Omron CX-Programmer project NewProject (CX-Programmer 9.87)

# PLC NewPLC1: CP1L M
; 

## Global symbols (name address type ; comment)
Banco_de_Dados_29 Contador_de_Peças_PH29
Banco_de_Dados_30 Contador_de_Peças_PH30
Banco_de_Dados_31 Contador_de_Peças_PH31
Conta_Peças Contador_de_Peças_PH31
PH11 0.03 BOOL
PH29 0.05 BOOL
PH30 0.04 BOOL
Visual_Formato_Trabalho_29 Formato_de_Trabalho_29
Visual_Formato_Trabalho_30 Formato_de_Trabalho_30
Visual_Formato_Trabalho_31 Formato_de_Trabalho_31
xx Formato_de_Trabalho_29

## Program NuovoProgramma1 (cyclic task 0)
Local symbols
F_31dias_vezes_2_ph30 D546 WORD
F_31dias_vezes_2_ph31 D530 WORD
F_Memoria_contagem_BCD_ph30 D552 WORD
F_Memoria_contagem_BCD_ph31 D536 WORD
F_Memória_de_Armazenagem_ph30 D550 WORD
F_Memória_de_Armazenagem_ph31 D534 WORD
F_Ponteiro_Dword_ph30 D548 WORD
F_Ponteiro_Dword_ph31 D532 WORD
KEEP 10.04 BOOL
MemAtuaReloSupervisorio H10.01 BOOL  ; Memória Atualiza Relogio pelo supervisório
Memoria_contagem_BCD_ph29 D528 WORD
Memoria_contagem_BCD_ph30 D518 WORD
Memoria_contagem_BCD_ph31 D508 WORD
Memoria_contagem_BIN_ph29 D526 WORD
Memoria_contagem_BIN_ph30 D516 WORD
Memoria_contagem_BIN_ph31 D506 WORD
Memória_de_Armazenagem_ph29 D524 WORD
Memória_de_Armazenagem_ph30 D514 WORD
Memória_de_Armazenagem_ph31 D504 WORD
PH29paradaT1 D0 CHANNEL  ; cnt prensa 31 parada T1
PH29paradaT2 D6 CHANNEL  ; cnt prensa 31 parada T2
PH29paradaT3 D12 CHANNEL  ; cnt prensa 31 parada T3
PH30paradaT1 D2 CHANNEL  ; cnt prensa 31 parada T1
PH30paradaT2 D8 CHANNEL  ; cnt prensa 31 parada T2
PH30paradaT3 D14 CHANNEL  ; cnt prensa 31 parada T3
PH31paradaT1 D4 CHANNEL  ; cnt prensa 31 parada T1
PH31paradaT2 D10 CHANNEL  ; cnt prensa 31 parada T2
PH31paradaT3 D18 CHANNEL  ; cnt prensa 31 parada T3
Ponteiro_Dword_ph29 D522 WORD
Ponteiro_Dword_ph30 D512 WORD
Ponteiro_Dword_ph31 D502 WORD
_31dias_vezes_2_ph29 D520 WORD
_31dias_vezes_2_ph30 D510 WORD
_31dias_vezes_2_ph31 D500 WORD
anoRelogio D36 CHANNEL  ; Ano Relógio
codFormPH29 D54 CHANNEL  ; Codigo do formato ph29
codFormPH30 D50 CHANNEL  ; Codigo do formato ph30
codFormPH31 D46 CHANNEL  ; Codigo do formato ph31
delayCicloPrensa29 T0001 BOOL  ; Retardo ciclo da prensa
delayCicloPrensa30 T0002 BOOL  ; Retardo ciclo da prensa
delayCicloPrensa31 T0003 BOOL  ; Retardo ciclo da prensa
diaCalendario D64 CHANNEL  ; dia calendario
diaMes D40 CHANNEL  ; dia do mes
diaRelogio D32 CHANNEL  ; Dia Relógio
filtroCntPc29 T0004 BOOL  ; filtro contagem peças
filtroCntPc30 T0005 BOOL  ; filtro contagem peças
filtroCntPc31 T0006 BOOL  ; filtro contagem peças
firstDMenvioFormat D56 CHANNEL  ; primeiro DM envio formato
firstDMenvioPcPH D42 CHANNEL  ; pirmeiro DM de envio peças ph
horaRelogio D30 CHANNEL  ; Horas Relogio
horas D58 CHANNEL  ; horas
iniciaCntTurno1 H10.02 BOOL  ; inicia contagem turno 1
iniciaCntTurno2 H10.03 BOOL  ; inicia contagem turno 2
iniciaCntTurno3 H10.04 BOOL  ; iniio contagem turno 3
linhaSelect D70 CHANNEL  ; linha selecionada
mesCalendario D66 CHANNEL  ; mes calendario
mesRelogio D34 CHANNEL  ; Mes Relogio
mesSelecionado D68 CHANNEL  ; mês selecionado
mesSelect D72 CHANNEL  ; mês selecionado
minutos D60 CHANNEL  ; minutos
minutosRelogio D28 CHANNEL  ; Minutos Relógio
numberCavidPH29 D52 CHANNEL  ; Número cavidades na prensa29
numberCavidPH30 D48 CHANNEL  ; Número cavidades na prensa30
numberCavidPH31 D44 CHANNEL  ; Número cavidades na prensa31
pecaPH29 D20 CHANNEL  ; conta peças ph29
pecaPH30 D22 CHANNEL  ; conta peças ph30
pecaPH31 D24 CHANNEL  ; conta peças ph31
ph29parada 10.00 BOOL  ; prensa 29 parada
ph30parada 10.01 BOOL  ; prensa 30 parada
ph31parada 10.03 BOOL  ; prensa 31 parada
ponteiroBDph29 D528 WORD  ; ponteiro banco de dados PH 29
ponteiroBDph30 D518 CHANNEL  ; ponteiro em BCD para armazenar a contagem
ponteiroBDph31 D508 WORD  ; ponteiro banco de dados PH31
prensa29 0.02 BOOL  ; Prensa 29
prensa30 0.01 BOOL  ; Prensa 30
prensa31 0.00 BOOL  ; Prensa 31
relogio4dig D38 CHANNEL  ; Ano Relógio 4 digitos
segundos D62 CHANNEL  ; segundos
segundosRelogio D26 CHANNEL  ; Segundos Relógio

### Section Reset

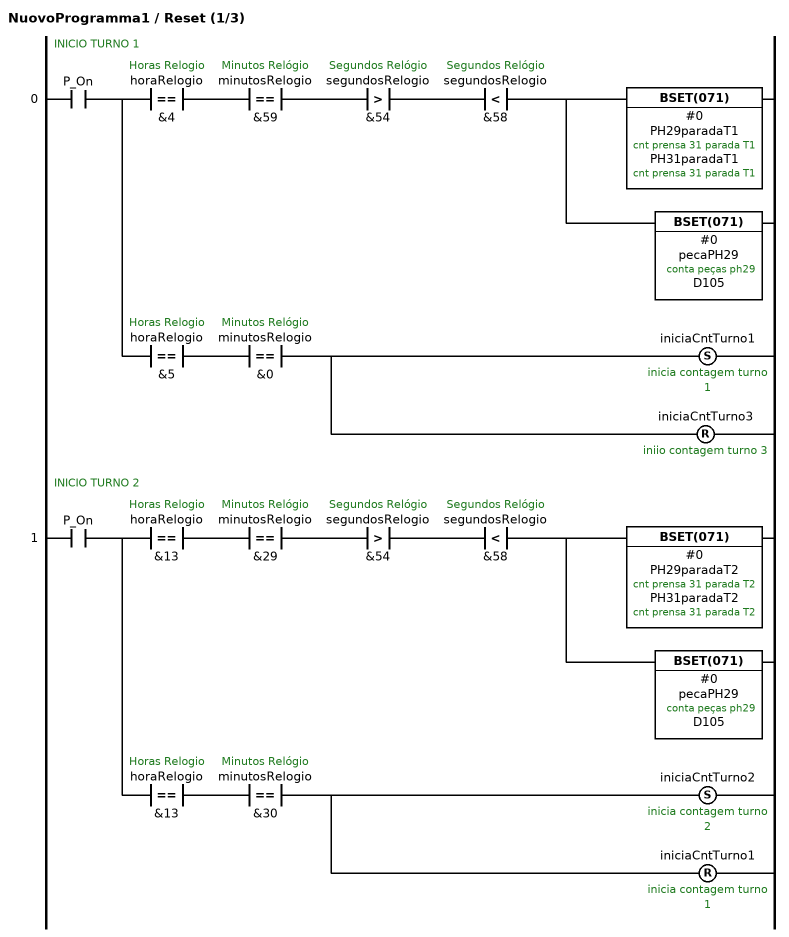
; rung 0: INICIO TURNO 1
LD P_On
OUT TR0
AND=(300) horaRelogio &4  ; Horas Relogio
AND=(300) minutosRelogio &59  ; Minutos Relógio
AND>(320) segundosRelogio &54  ; Segundos Relógio
AND<(310) segundosRelogio &58  ; Segundos Relógio
BSET(071) #0 PH29paradaT1 PH31paradaT1  ; cnt prensa 31 parada T1
BSET(071) #0 pecaPH29 D105  ; conta peças ph29
LD TR0
AND=(300) horaRelogio &5  ; Horas Relogio
AND=(300) minutosRelogio &0  ; Minutos Relógio
SET iniciaCntTurno1  ; inicia contagem turno 1
RSET iniciaCntTurno3  ; iniio contagem turno 3
; rung 1: INICIO TURNO 2
LD P_On
OUT TR0
AND=(300) horaRelogio &13  ; Horas Relogio
AND=(300) minutosRelogio &29  ; Minutos Relógio
AND>(320) segundosRelogio &54  ; Segundos Relógio
AND<(310) segundosRelogio &58  ; Segundos Relógio
BSET(071) #0 PH29paradaT2 PH31paradaT2  ; cnt prensa 31 parada T2
BSET(071) #0 pecaPH29 D105  ; conta peças ph29
LD TR0
AND=(300) horaRelogio &13  ; Horas Relogio
AND=(300) minutosRelogio &30  ; Minutos Relógio
SET iniciaCntTurno2  ; inicia contagem turno 2
RSET iniciaCntTurno1  ; inicia contagem turno 1

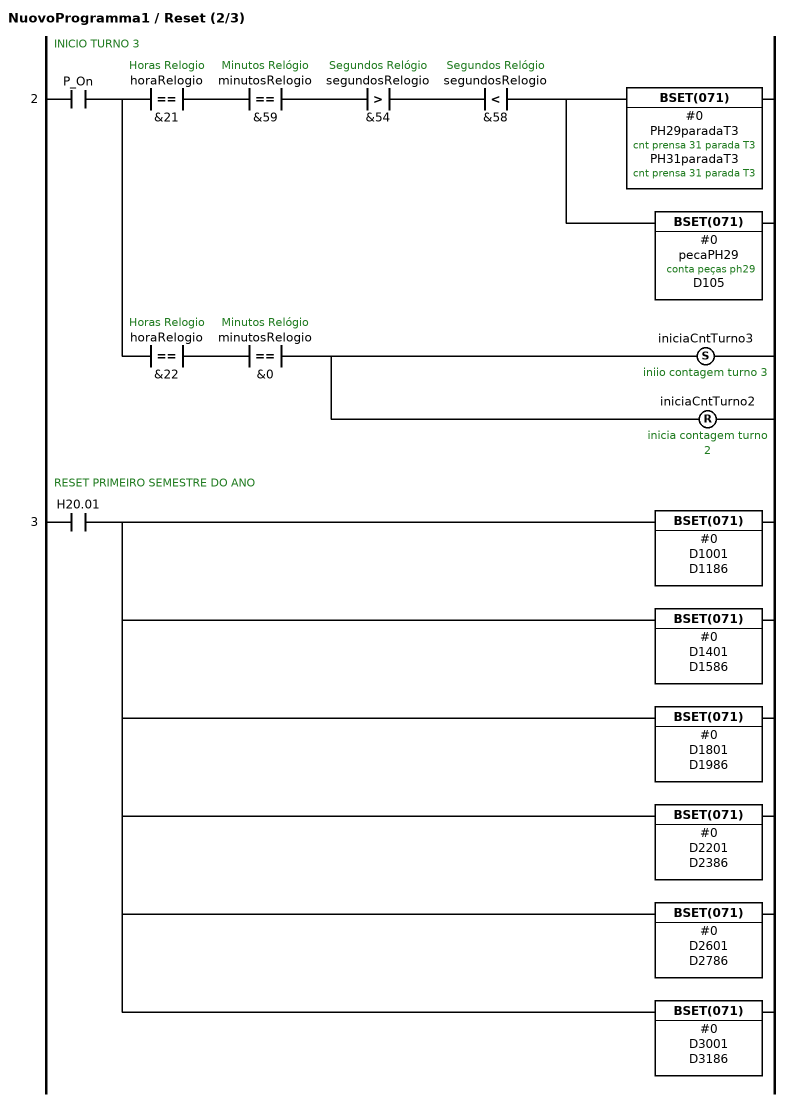
; rung 2: INICIO TURNO 3
LD P_On
OUT TR0
AND=(300) horaRelogio &21  ; Horas Relogio
AND=(300) minutosRelogio &59  ; Minutos Relógio
AND>(320) segundosRelogio &54  ; Segundos Relógio
AND<(310) segundosRelogio &58  ; Segundos Relógio
BSET(071) #0 PH29paradaT3 PH31paradaT3  ; cnt prensa 31 parada T3
BSET(071) #0 pecaPH29 D105  ; conta peças ph29
LD TR0
AND=(300) horaRelogio &22  ; Horas Relogio
AND=(300) minutosRelogio &0  ; Minutos Relógio
SET iniciaCntTurno3  ; iniio contagem turno 3
RSET iniciaCntTurno2  ; inicia contagem turno 2
; rung 3: RESET PRIMEIRO SEMESTRE DO ANO
LD H20.01
BSET(071) #0 D1001 D1186  // RESET PH31, 01/01 ATÉ 31/06
BSET(071) #0 D1401 D1586  // RESET PH30, 01/01 ATÉ 31/06
BSET(071) #0 D1801 D1986  // RESET PH29, 01/01 ATÉ 31/06
BSET(071) #0 D2201 D2386  // RESET FORMATO PH31, 01/01 ATÉ 31/06
BSET(071) #0 D2601 D2786  // RESET FORMATO PH30, 01/01 ATÉ 31/06
BSET(071) #0 D3001 D3186  // RESET FORMATO PH29, 01/01 ATÉ 31/06

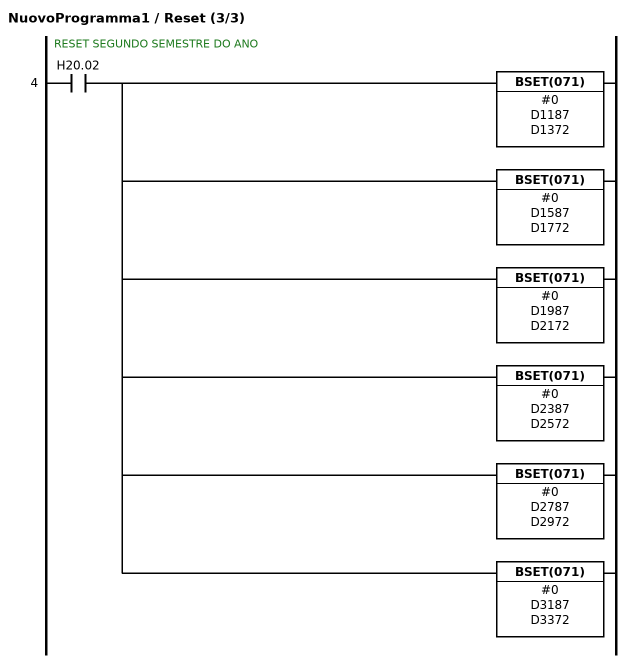
; rung 4: RESET SEGUNDO SEMESTRE DO ANO
LD H20.02
BSET(071) #0 D1187 D1372  // RESET PH31, 01/07 ATÉ 31/12
BSET(071) #0 D1587 D1772  // RESET PH30, 01/07 ATÉ 31/12
BSET(071) #0 D1987 D2172  // RESET PH29, 01/07 ATÉ 31/12
BSET(071) #0 D2387 D2572  // RESET FORMATO PH31, 01/07 ATÉ 31/12
BSET(071) #0 D2787 D2972  // RESET FORMATO PH30, 01/07 ATÉ 31/12
BSET(071) #0 D3187 D3372  // RESET FORMATO PH29, 01/07 ATÉ 31/12

### Section PH29

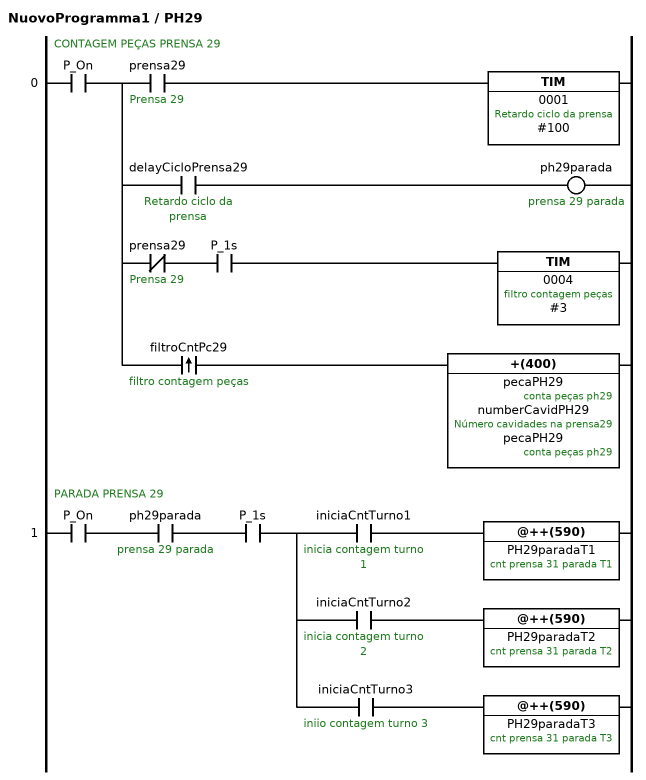
; rung 0: CONTAGEM PEÇAS PRENSA 29
LD P_On
OUT TR0
AND prensa29  ; Prensa 29
TIM 0001 #100  ; Retardo ciclo da prensa
LD TR0
AND delayCicloPrensa29  ; Retardo ciclo da prensa
OUT ph29parada  ; prensa 29 parada
LD TR0
ANDNOT prensa29  ; Prensa 29
AND P_1s
TIM 0004 #3  ; filtro contagem peças
LD TR0
@AND filtroCntPc29  ; filtro contagem peças
+(400) pecaPH29 numberCavidPH29 pecaPH29  ; conta peças ph29, Número cavidades na prensa29
; rung 1: PARADA PRENSA 29
LD P_On
AND ph29parada  ; prensa 29 parada
AND P_1s
OUT TR0
AND iniciaCntTurno1  ; inicia contagem turno 1
@++(590) PH29paradaT1  ; cnt prensa 31 parada T1  // CONTA PARADA TURNO 1
LD TR0
AND iniciaCntTurno2  ; inicia contagem turno 2
@++(590) PH29paradaT2  ; cnt prensa 31 parada T2  // CONTA PARADA TURNO 2
LD TR0
AND iniciaCntTurno3  ; iniio contagem turno 3
@++(590) PH29paradaT3  ; cnt prensa 31 parada T3  // CONTA PARADA TURNO 3

### Section PH30

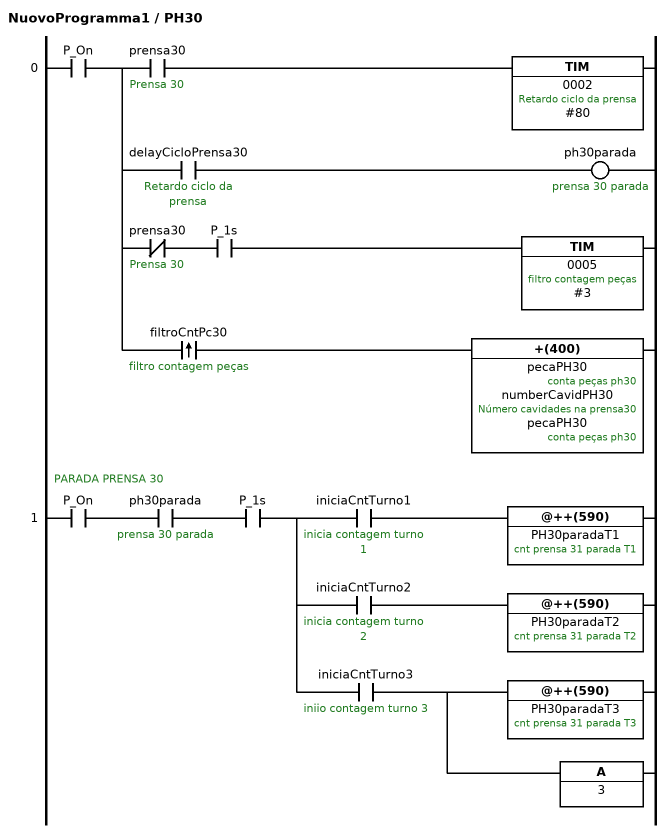
; rung 0
LD P_On
OUT TR0
AND prensa30  ; Prensa 30
TIM 0002 #80  ; Retardo ciclo da prensa
LD TR0
AND delayCicloPrensa30  ; Retardo ciclo da prensa
OUT ph30parada  ; prensa 30 parada
LD TR0
ANDNOT prensa30  ; Prensa 30
AND P_1s
TIM 0005 #3  ; filtro contagem peças
LD TR0
@AND filtroCntPc30  ; filtro contagem peças
+(400) pecaPH30 numberCavidPH30 pecaPH30  ; conta peças ph30, Número cavidades na prensa30
; rung 1: PARADA PRENSA 30
LD P_On  // D20 CONTA TURNO 2
AND ph30parada  ; prensa 30 parada
AND P_1s
OUT TR0
AND iniciaCntTurno1  ; inicia contagem turno 1
@++(590) PH30paradaT1  ; cnt prensa 31 parada T1  // 
LD TR0
AND iniciaCntTurno2  ; inicia contagem turno 2
@++(590) PH30paradaT2  ; cnt prensa 31 parada T2
LD TR0
AND iniciaCntTurno3  ; iniio contagem turno 3
@++(590) PH30paradaT3  ; cnt prensa 31 parada T3  // D18 CONTA TURNO 1
A  3
// D22 CONTA TURNO 3

### Section PH31

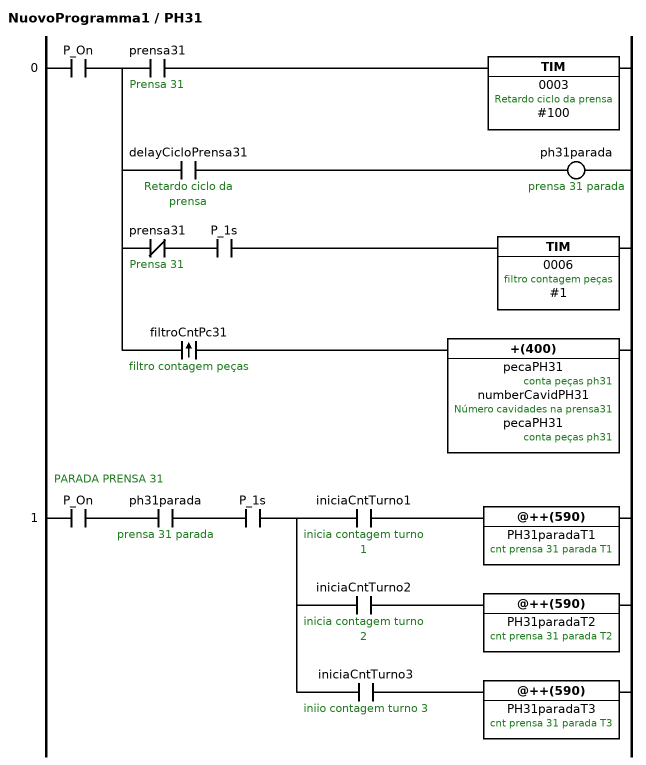
; rung 0
LD P_On
OUT TR0
AND prensa31  ; Prensa 31
TIM 0003 #100  ; Retardo ciclo da prensa
LD TR0
AND delayCicloPrensa31  ; Retardo ciclo da prensa
OUT ph31parada  ; prensa 31 parada
LD TR0
ANDNOT prensa31  ; Prensa 31
AND P_1s
TIM 0006 #1  ; filtro contagem peças
LD TR0
@AND filtroCntPc31  ; filtro contagem peças
+(400) pecaPH31 numberCavidPH31 pecaPH31  ; conta peças ph31, Número cavidades na prensa31
; rung 1: PARADA PRENSA 31
LD P_On
AND ph31parada  ; prensa 31 parada
AND P_1s
OUT TR0
AND iniciaCntTurno1  ; inicia contagem turno 1
@++(590) PH31paradaT1  ; cnt prensa 31 parada T1  // CONTA PARADA TURNO 1
LD TR0
AND iniciaCntTurno2  ; inicia contagem turno 2
@++(590) PH31paradaT2  ; cnt prensa 31 parada T2  // CONTA PARADA TURNO 2
LD TR0
AND iniciaCntTurno3  ; iniio contagem turno 3
@++(590) PH31paradaT3  ; cnt prensa 31 parada T3  // CONTA PARADA TUNOR 3

### Section Banco_de_Dados

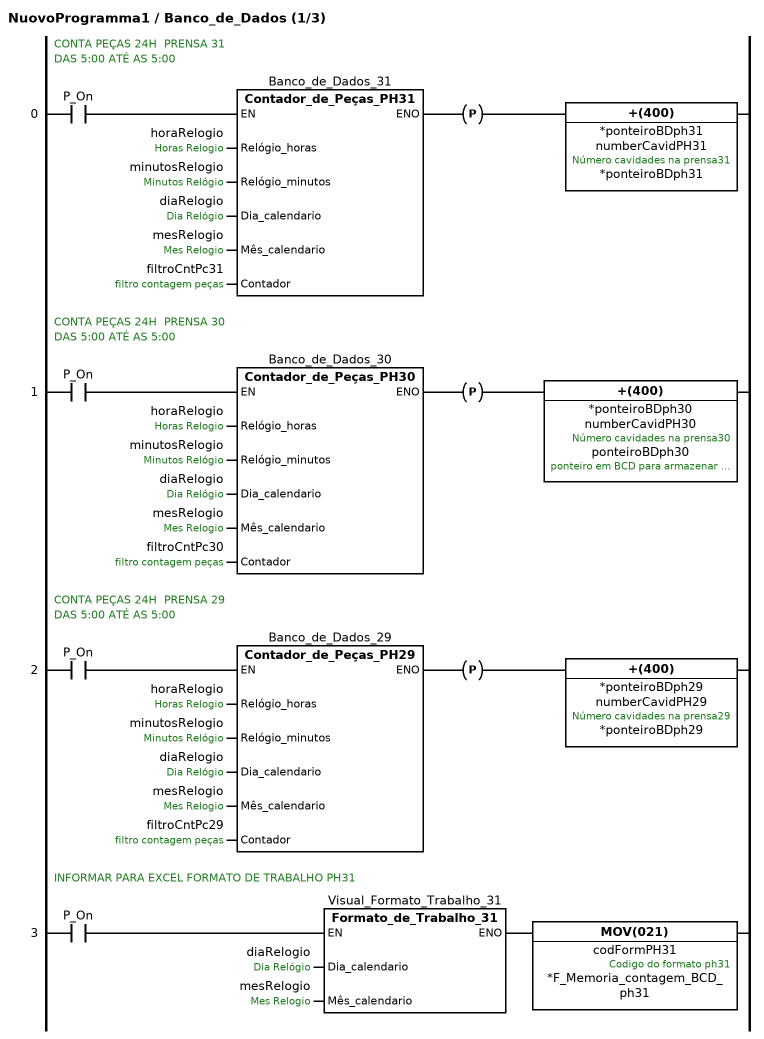
; rung 0: CONTA PEÇAS 24H  PRENSA 31 / DAS 5:00 ATÉ AS 5:00
LD P_On
CALL Banco_de_Dados_31 : Contador_de_Peças_PH31 (Relógio_horas := horaRelogio, Relógio_minutos := minutosRelogio, Dia_calendario := diaRelogio, Mês_calendario := mesRelogio, Contador := filtroCntPc31)  ; Horas Relogio, Minutos Relógio, Dia Relógio, Mes Relogio, filtro contagem peças
UP(521)
+(400) *ponteiroBDph31 numberCavidPH31 *ponteiroBDph31  ; Número cavidades na prensa31
; rung 1: CONTA PEÇAS 24H  PRENSA 30 / DAS 5:00 ATÉ AS 5:00
LD P_On
CALL Banco_de_Dados_30 : Contador_de_Peças_PH30 (Relógio_horas := horaRelogio, Relógio_minutos := minutosRelogio, Dia_calendario := diaRelogio, Mês_calendario := mesRelogio, Contador := filtroCntPc30)  ; Horas Relogio, Minutos Relógio, Dia Relógio, Mes Relogio, filtro contagem peças
UP(521)
+(400) *ponteiroBDph30 numberCavidPH30 ponteiroBDph30  ; Número cavidades na prensa30, ponteiro em BCD para armazenar a contagem
; rung 2: CONTA PEÇAS 24H  PRENSA 29 / DAS 5:00 ATÉ AS 5:00
LD P_On
CALL Banco_de_Dados_29 : Contador_de_Peças_PH29 (Relógio_horas := horaRelogio, Relógio_minutos := minutosRelogio, Dia_calendario := diaRelogio, Mês_calendario := mesRelogio, Contador := filtroCntPc29)  ; Horas Relogio, Minutos Relógio, Dia Relógio, Mes Relogio, filtro contagem peças
UP(521)
+(400) *ponteiroBDph29 numberCavidPH29 *ponteiroBDph29  ; Número cavidades na prensa29
; rung 3: INFORMAR PARA EXCEL FORMATO DE TRABALHO PH31
LD P_On
CALL Visual_Formato_Trabalho_31 : Formato_de_Trabalho_31 (Dia_calendario := diaRelogio, Mês_calendario := mesRelogio)  ; Dia Relógio, Mes Relogio
MOV(021) codFormPH31 *F_Memoria_contagem_BCD_ph31  ; Codigo do formato ph31

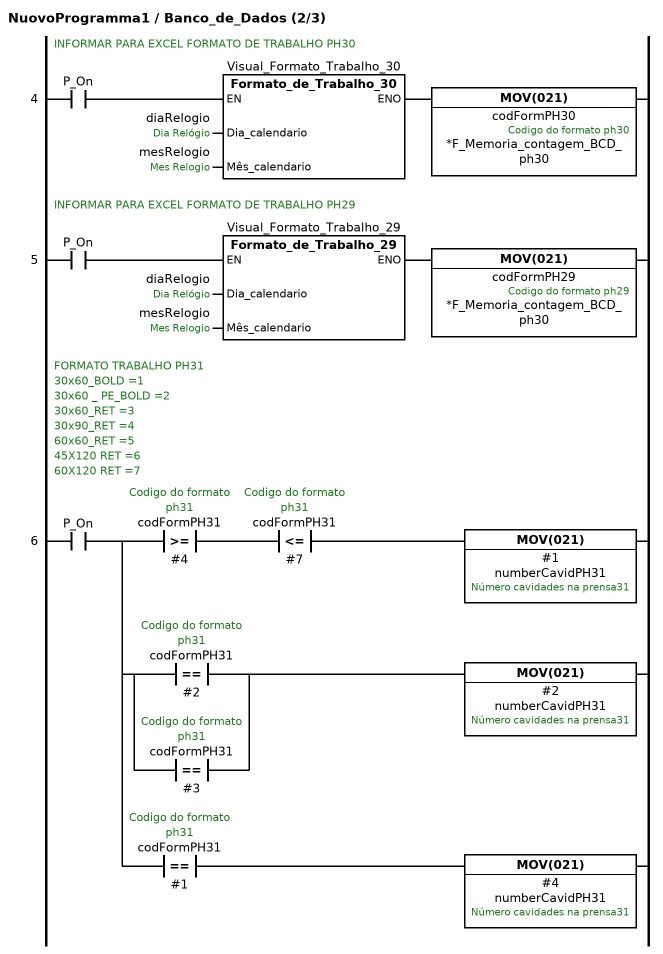
; rung 4: INFORMAR PARA EXCEL FORMATO DE TRABALHO PH30
LD P_On
CALL Visual_Formato_Trabalho_30 : Formato_de_Trabalho_30 (Dia_calendario := diaRelogio, Mês_calendario := mesRelogio)  ; Dia Relógio, Mes Relogio
MOV(021) codFormPH30 *F_Memoria_contagem_BCD_ph30  ; Codigo do formato ph30
; rung 5: INFORMAR PARA EXCEL FORMATO DE TRABALHO PH29
LD P_On
CALL Visual_Formato_Trabalho_29 : Formato_de_Trabalho_29 (Dia_calendario := diaRelogio, Mês_calendario := mesRelogio)  ; Dia Relógio, Mes Relogio
MOV(021) codFormPH29 *F_Memoria_contagem_BCD_ph30  ; Codigo do formato ph29
; rung 6: FORMATO TRABALHO PH31 / 30x60_BOLD =1 / 30x60_PE_BOLD =2 / 30x60_RET =3 / 30x90_RET =4 / 60x60_RET =5 / 45X120 RET =6 / 60X120 RET =7
LD P_On
OUT TR0
AND>=(325) codFormPH31 #4  ; Codigo do formato ph31
AND<=(315) codFormPH31 #7  ; Codigo do formato ph31
MOV(021) #1 numberCavidPH31  ; Número cavidades na prensa31
LD TR0
LD=(300) codFormPH31 #2  ; Codigo do formato ph31
OR=(300) codFormPH31 #3  ; Codigo do formato ph31
ANDLD
MOV(021) #2 numberCavidPH31  ; Número cavidades na prensa31
LD TR0
AND=(300) codFormPH31 #1  ; Codigo do formato ph31
MOV(021) #4 numberCavidPH31  ; Número cavidades na prensa31

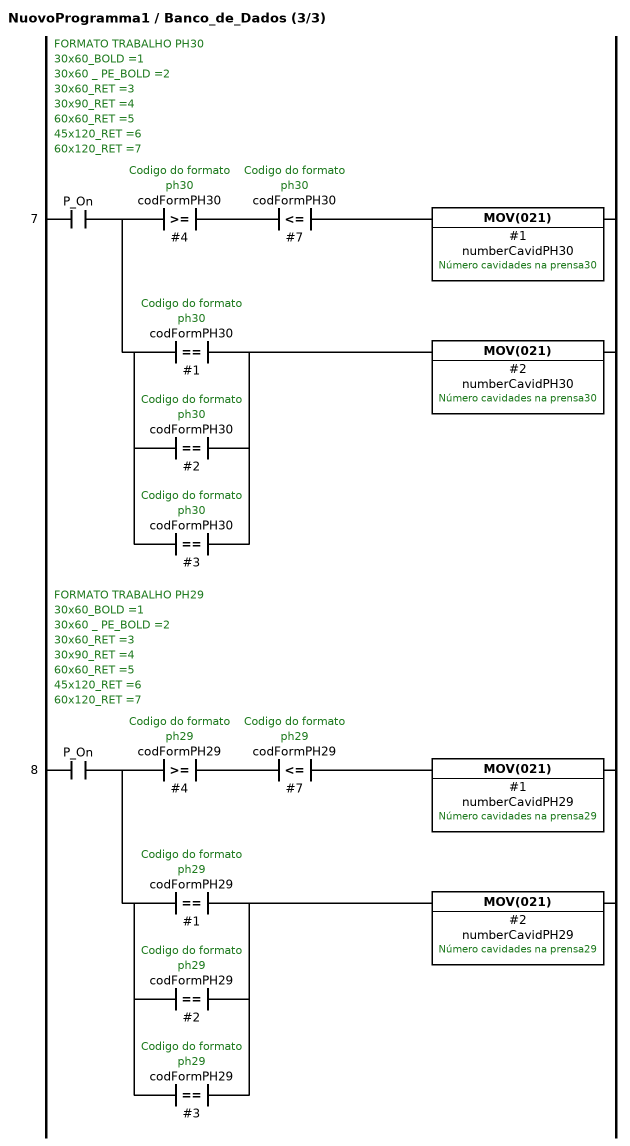
; rung 7: FORMATO TRABALHO PH30 / 30x60_BOLD =1 / 30x60_PE_BOLD =2 / 30x60_RET =3 / 30x90_RET =4 / 60x60_RET =5 / 45x120_RET =6 / 60x120_RET =7
LD P_On
OUT TR0
AND>=(325) codFormPH30 #4  ; Codigo do formato ph30
AND<=(315) codFormPH30 #7  ; Codigo do formato ph30
MOV(021) #1 numberCavidPH30  ; Número cavidades na prensa30
LD TR0
LD=(300) codFormPH30 #1  ; Codigo do formato ph30
OR=(300) codFormPH30 #2  ; Codigo do formato ph30
OR=(300) codFormPH30 #3  ; Codigo do formato ph30
ANDLD
MOV(021) #2 numberCavidPH30  ; Número cavidades na prensa30
; rung 8: FORMATO TRABALHO PH29 / 30x60_BOLD =1 / 30x60_PE_BOLD =2 / 30x60_RET =3 / 30x90_RET =4 / 60x60_RET =5 / 45x120_RET =6 / 60x120_RET =7
LD P_On
OUT TR0
AND>=(325) codFormPH29 #4  ; Codigo do formato ph29
AND<=(315) codFormPH29 #7  ; Codigo do formato ph29
MOV(021) #1 numberCavidPH29  ; Número cavidades na prensa29
LD TR0
LD=(300) codFormPH29 #1  ; Codigo do formato ph29
OR=(300) codFormPH29 #2  ; Codigo do formato ph29
OR=(300) codFormPH29 #3  ; Codigo do formato ph29
ANDLD
MOV(021) #2 numberCavidPH29  ; Número cavidades na prensa29

### Section Transferencia_excel

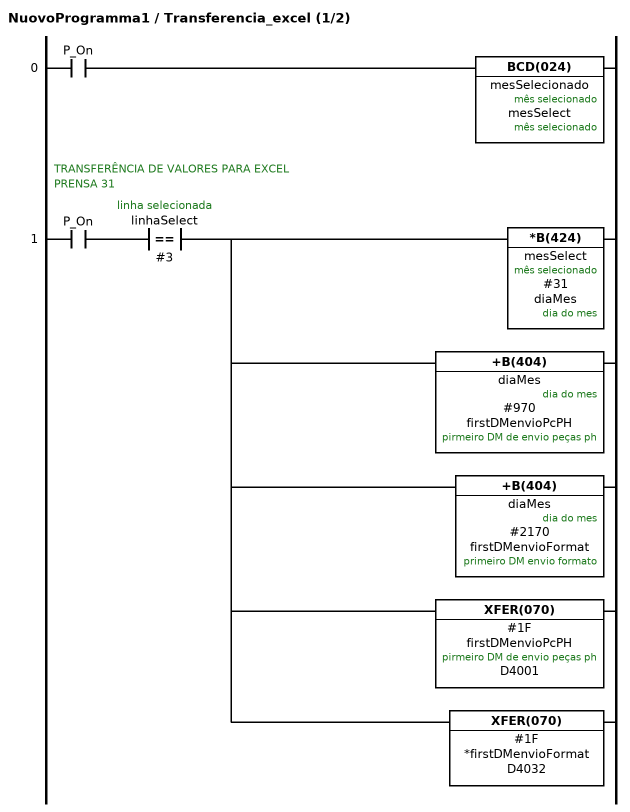
; rung 0
LD P_On
BCD(024) mesSelecionado mesSelect  ; mês selecionado
; rung 1: TRANSFERÊNCIA DE VALORES PARA EXCEL / PRENSA 31
LD P_On
AND=(300) linhaSelect #3  ; linha selecionada
*B(424) mesSelect #31 diaMes  ; mês selecionado, dia do mes  // SELECIONA O MES MULTIPLICA POR 31
+B(404) diaMes #970 firstDMenvioPcPH  ; dia do mes, pirmeiro DM de envio peças ph  // NUMERO DE DIAS DO ANO MULTIPLICA 970
+B(404) diaMes #2170 firstDMenvioFormat  ; dia do mes, primeiro DM envio formato
XFER(070) #1F firstDMenvioPcPH D4001  ; pirmeiro DM de envio peças ph  // TRANSFERE 31 DM APARTIR DO PRIMEIRO DM DE ENVIO
XFER(070) #1F *firstDMenvioFormat D4032

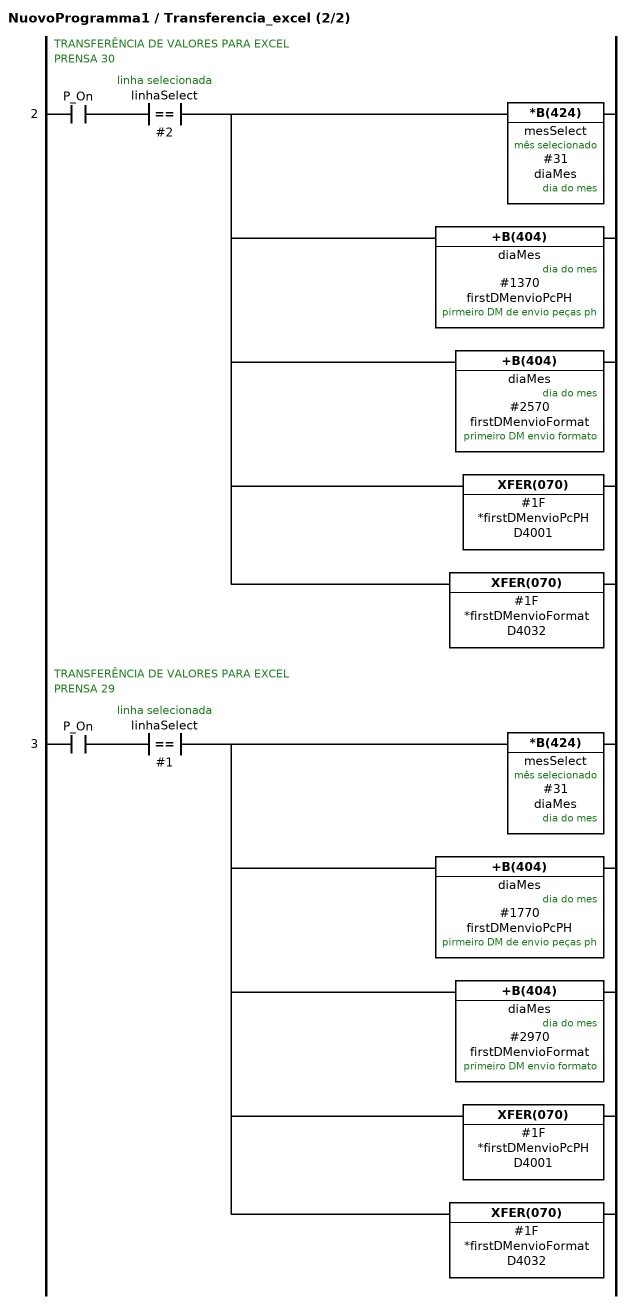
; rung 2: TRANSFERÊNCIA DE VALORES PARA EXCEL / PRENSA 30
LD P_On
AND=(300) linhaSelect #2  ; linha selecionada
*B(424) mesSelect #31 diaMes  ; mês selecionado, dia do mes
+B(404) diaMes #1370 firstDMenvioPcPH  ; dia do mes, pirmeiro DM de envio peças ph
+B(404) diaMes #2570 firstDMenvioFormat  ; dia do mes, primeiro DM envio formato
XFER(070) #1F *firstDMenvioPcPH D4001
XFER(070) #1F *firstDMenvioFormat D4032
; rung 3: TRANSFERÊNCIA DE VALORES PARA EXCEL / PRENSA 29
LD P_On
AND=(300) linhaSelect #1  ; linha selecionada
*B(424) mesSelect #31 diaMes  ; mês selecionado, dia do mes
+B(404) diaMes #1770 firstDMenvioPcPH  ; dia do mes, pirmeiro DM de envio peças ph
+B(404) diaMes #2970 firstDMenvioFormat  ; dia do mes, primeiro DM envio formato
XFER(070) #1F *firstDMenvioPcPH D4001
XFER(070) #1F *firstDMenvioFormat D4032

### Section Relogio

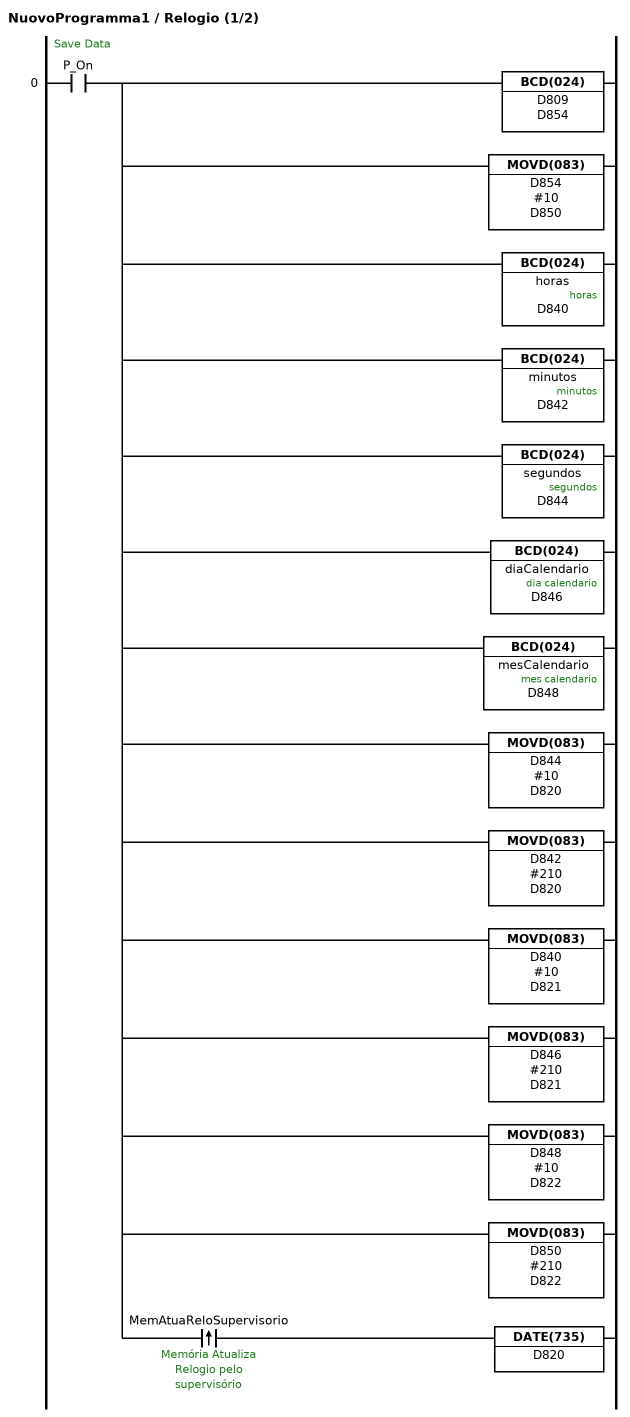
; rung 0: Save Data
LD P_On
BCD(024) D809 D854
MOVD(083) D854 #10 D850
BCD(024) horas D840  ; horas
BCD(024) minutos D842  ; minutos
BCD(024) segundos D844  ; segundos
BCD(024) diaCalendario D846  ; dia calendario
BCD(024) mesCalendario D848  ; mes calendario
MOVD(083) D844 #10 D820
MOVD(083) D842 #210 D820
MOVD(083) D840 #10 D821
MOVD(083) D846 #210 D821
MOVD(083) D848 #10 D822
MOVD(083) D850 #210 D822
@AND MemAtuaReloSupervisorio  ; Memória Atualiza Relogio pelo supervisório
DATE(735) D820

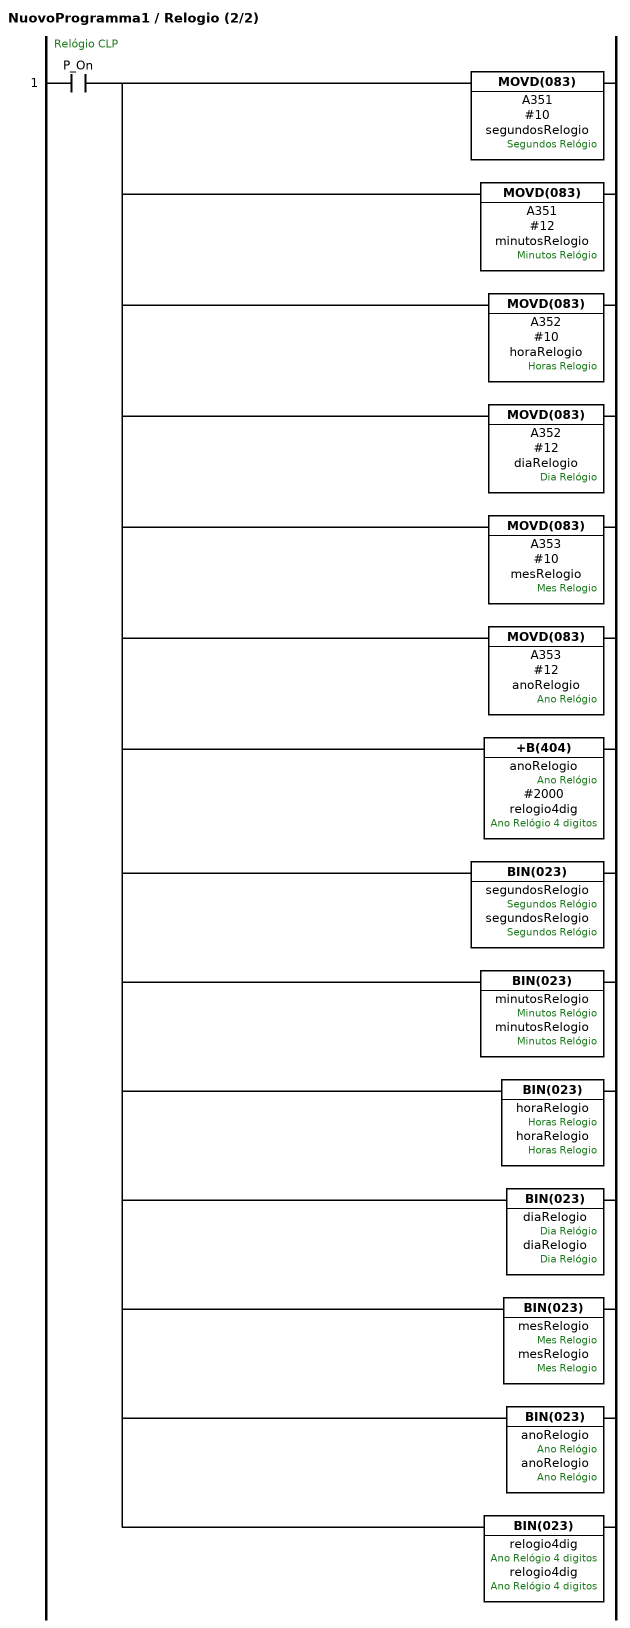
; rung 1: Relógio CLP
LD P_On
MOVD(083) A351 #10 segundosRelogio  ; Segundos Relógio
MOVD(083) A351 #12 minutosRelogio  ; Minutos Relógio
MOVD(083) A352 #10 horaRelogio  ; Horas Relogio
MOVD(083) A352 #12 diaRelogio  ; Dia Relógio
MOVD(083) A353 #10 mesRelogio  ; Mes Relogio
MOVD(083) A353 #12 anoRelogio  ; Ano Relógio
+B(404) anoRelogio #2000 relogio4dig  ; Ano Relógio, Ano Relógio 4 digitos
BIN(023) segundosRelogio segundosRelogio  ; Segundos Relógio
BIN(023) minutosRelogio minutosRelogio  ; Minutos Relógio
BIN(023) horaRelogio horaRelogio  ; Horas Relogio
BIN(023) diaRelogio diaRelogio  ; Dia Relógio
BIN(023) mesRelogio mesRelogio  ; Mes Relogio
BIN(023) anoRelogio anoRelogio  ; Ano Relógio
BIN(023) relogio4dig relogio4dig  ; Ano Relógio 4 digitos

### Section END
; rung 0
END(001)

## Function block Contador_de_Peças_PH29
VAR_INPUT
  Relógio_horas : WORD;
  Relógio_minutos : WORD;
  Dia_calendario : WORD;
  Mês_calendario : WORD;
  Contador : BOOL;
END_VAR
VAR
  _31dias_vezes_2 AT D520 : WORD;
  Ponteiro_DWord AT D522 : WORD;
  Memória_de_Armazenagem AT D524 : WORD;
  Memoria_contagem_BIN AT D526 : WORD;
  Memoria_contagem_BCD AT D528 : WORD;
END_VAR

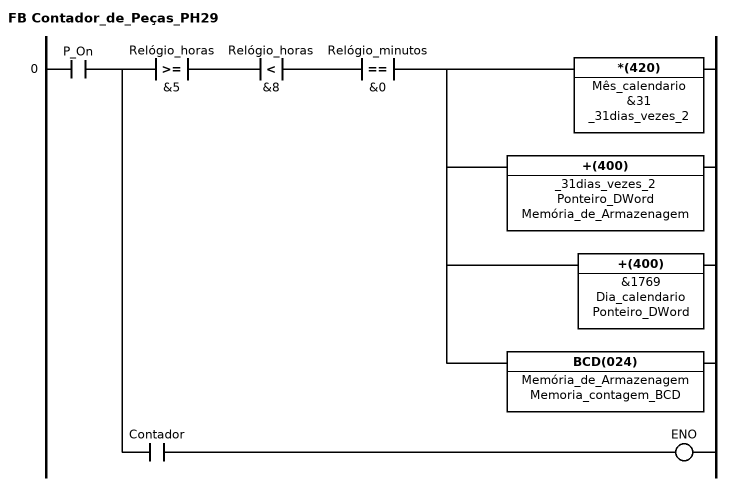
; rung 0
LD P_On
OUT TR0
AND>=(325) Relógio_horas &5
AND<(310) Relógio_horas &8
AND=(300) Relógio_minutos &0
*(420) Mês_calendario &31 _31dias_vezes_2
+(400) _31dias_vezes_2 Ponteiro_DWord Memória_de_Armazenagem
+(400) &1769 Dia_calendario Ponteiro_DWord
BCD(024) Memória_de_Armazenagem Memoria_contagem_BCD
LD TR0
AND Contador
OUT ENO

## Function block Contador_de_Peças_PH30
VAR_INPUT
  Relógio_horas : WORD;
  Relógio_minutos : WORD;
  Dia_calendario : WORD;
  Mês_calendario : WORD;
  Contador : BOOL;
END_VAR
VAR
  _31dias_vezes_2 AT D510 : WORD;
  Ponteiro_DWord AT D512 : WORD;
  Memória_de_Armazenagem AT D514 : WORD;
  Memoria_contagem_BIN AT D516 : WORD;
  Memoria_contagem_BCD AT D518 : WORD;
END_VAR

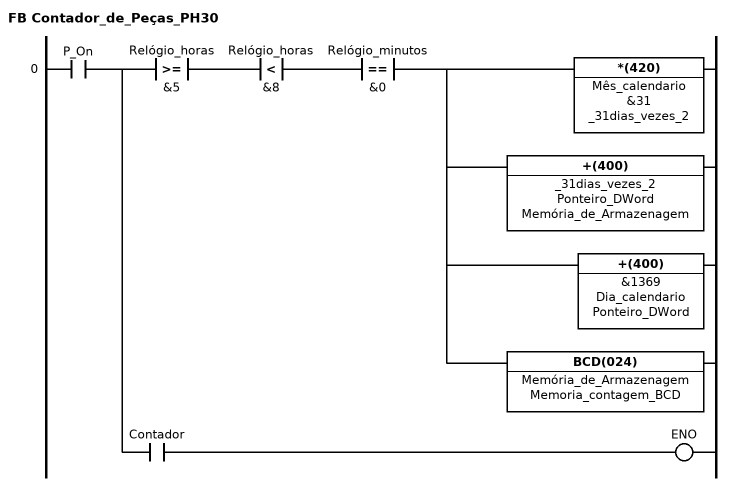
; rung 0
LD P_On
OUT TR0
AND>=(325) Relógio_horas &5
AND<(310) Relógio_horas &8
AND=(300) Relógio_minutos &0
*(420) Mês_calendario &31 _31dias_vezes_2
+(400) _31dias_vezes_2 Ponteiro_DWord Memória_de_Armazenagem
+(400) &1369 Dia_calendario Ponteiro_DWord
BCD(024) Memória_de_Armazenagem Memoria_contagem_BCD
LD TR0
AND Contador
OUT ENO

## Function block Contador_de_Peças_PH31
VAR_INPUT
  Relógio_horas : WORD;
  Relógio_minutos : WORD;
  Dia_calendario : WORD;
  Mês_calendario : WORD;
  Contador : BOOL;
END_VAR
VAR
  _31dias_vezes_2 AT D500 : WORD;
  Ponteiro_DWord AT D502 : WORD;
  Memória_de_Armazenagem AT D504 : WORD;
  Memoria_contagem_BIN AT D506 : WORD;
  Memoria_contagem_BCD AT D508 : WORD;
END_VAR

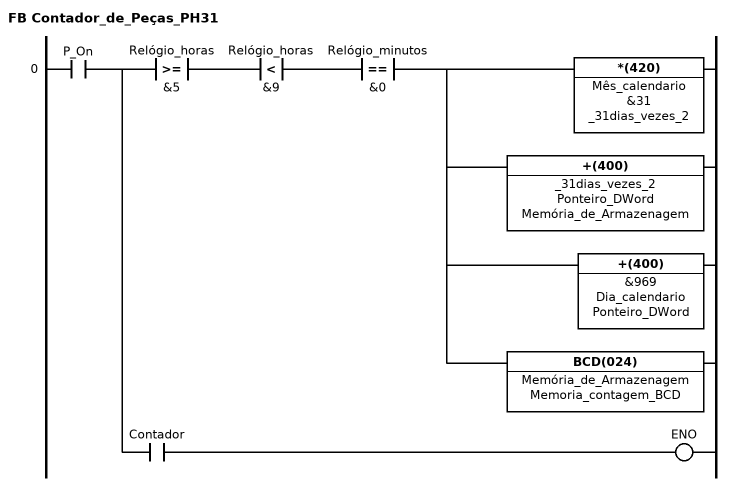
; rung 0
LD P_On
OUT TR0
AND>=(325) Relógio_horas &5
AND<(310) Relógio_horas &9
AND=(300) Relógio_minutos &0
*(420) Mês_calendario &31 _31dias_vezes_2
+(400) _31dias_vezes_2 Ponteiro_DWord Memória_de_Armazenagem
+(400) &969 Dia_calendario Ponteiro_DWord
BCD(024) Memória_de_Armazenagem Memoria_contagem_BCD
LD TR0
AND Contador
OUT ENO

## Function block Formato_de_Trabalho_29
VAR_INPUT
  Dia_calendario : WORD;
  Mês_calendario : WORD;
END_VAR
VAR
  _31dias_vezes_2 AT D546 : WORD;
  Ponteiro_DWord AT D548 : WORD;
  Memória_de_Armazenagem AT D550 : WORD;
  Memoria_contagem_BCD AT D552 : WORD;
END_VAR

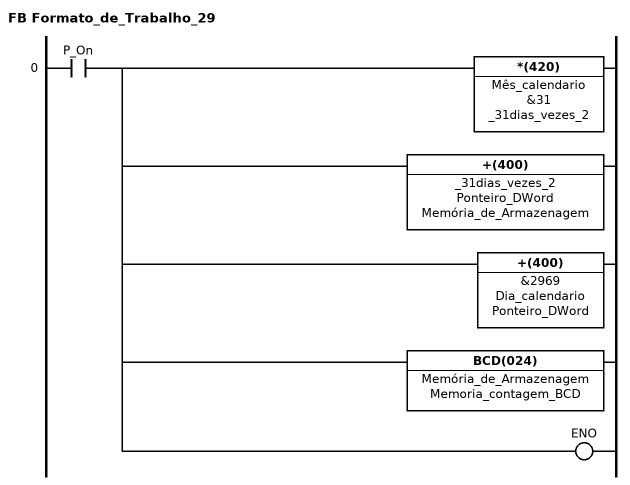
; rung 0
LD P_On
*(420) Mês_calendario &31 _31dias_vezes_2
+(400) _31dias_vezes_2 Ponteiro_DWord Memória_de_Armazenagem
+(400) &2969 Dia_calendario Ponteiro_DWord
BCD(024) Memória_de_Armazenagem Memoria_contagem_BCD
OUT ENO

## Function block Formato_de_Trabalho_30
VAR_INPUT
  Dia_calendario : WORD;
  Mês_calendario : WORD;
END_VAR
VAR
  _31dias_vezes_2 AT D538 : WORD;
  Ponteiro_DWord AT D540 : WORD;
  Memória_de_Armazenagem AT D542 : WORD;
  Memoria_contagem_BCD AT D544 : WORD;
END_VAR

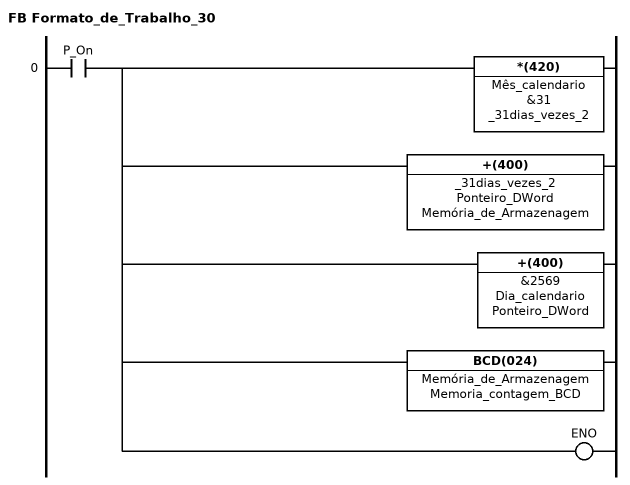
; rung 0
LD P_On
*(420) Mês_calendario &31 _31dias_vezes_2
+(400) _31dias_vezes_2 Ponteiro_DWord Memória_de_Armazenagem
+(400) &2569 Dia_calendario Ponteiro_DWord
BCD(024) Memória_de_Armazenagem Memoria_contagem_BCD
OUT ENO

## Function block Formato_de_Trabalho_31
VAR_INPUT
  Dia_calendario : WORD;
  Mês_calendario : WORD;
END_VAR
VAR
  _31dias_vezes_2 AT D530 : WORD;
  Ponteiro_DWord AT D532 : WORD;
  Memória_de_Armazenagem AT D534 : WORD;
  Memoria_contagem_BCD AT D536 : WORD;
END_VAR

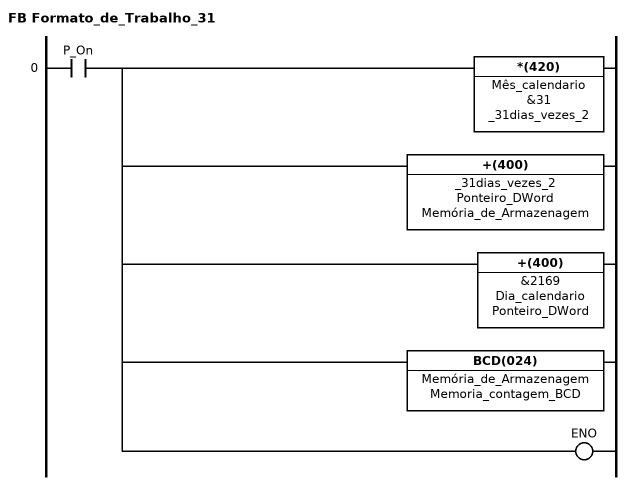
; rung 0
LD P_On
*(420) Mês_calendario &31 _31dias_vezes_2
+(400) _31dias_vezes_2 Ponteiro_DWord Memória_de_Armazenagem
+(400) &2169 Dia_calendario Ponteiro_DWord
BCD(024) Memória_de_Armazenagem Memoria_contagem_BCD
OUT ENO

# PLC NewPLC2: CPM1(CPM1A) CPU10

## Program NewProgram1 (no task)

### Section Section1

### Section END
; rung 0
END(01)